FUNCTION_BLOCK FB_ParameterList // store params for permanence. THEY MUST BE PART OF AN OBJECT ELSEWHERE!
VAR
	_unNumberOfEntries : UDINT;
	_unIndexForProperties : UDINT;
	asDictionary : ARRAY[0..MAX_DICTIONARY_SIZE] OF ST_KeyReferencePair;
END_VAR
VAR CONSTANT
	MAX_DICTIONARY_SIZE : UDINT := 1000; // arbitrary
END_VAR

METHOD PUBLIC AddToList : BOOL
VAR_INPUT
	sKey : T_MaxString;
	tRef : T_Arg;
END_VAR
IF KeyExists(sKey) THEN
	RETURN;
END_IF

IF _unNumberOfEntries + 1 > MAX_DICTIONARY_SIZE THEN
	RETURN;
END_IF

asDictionary[_unNumberOfEntries].Key := sKey;
asDictionary[_unNumberOfEntries].Ref := tRef;

_unNumberOfEntries := _unNumberOfEntries + 1;

AddToList := TRUE;
END_METHOD

METHOD PUBLIC ClearList
VAR 
	indexer : UDINT;
	sBlankKeyRef : ST_KeyReferencePair;
END_VAR
FOR indexer := 0 TO _unNumberOfEntries - 1 DO
	asDictionary[indexer] := sBlankKeyRef;
END_FOR

_unNumberOfEntries := 0;
END_METHOD

METHOD PUBLIC GetByKey : T_Arg
VAR_INPUT
	sKey : STRING;
END_VAR

VAR
	indexer : UDINT;
END_VAR
FOR indexer := 0 TO _unNumberOfEntries - 1 DO
	
	IF asDictionary[indexer].Key = sKey THEN
		GetByKey := asDictionary[indexer].Ref;
		RETURN;
	END_IF;
	
END_FOR
END_METHOD

PROPERTY PUBLIC Index : UDINT
GET
Index := _unIndexForProperties;
END_GET
SET
IF Index  < _unNumberOfEntries THEN
	_unIndexForProperties := Index;
ELSE
	_unIndexForProperties := _unNumberOfEntries;
END_IF
END_SET
END_PROPERTY

PROPERTY PRIVATE IndexKey : STRING
GET // PUBLIC
IF _unIndexForProperties < _unNumberOfEntries THEN
	IndexKey := asDictionary[_unIndexForProperties].Key;
END_IF;
END_GET
END_PROPERTY

PROPERTY PRIVATE IndexRef : T_Arg
GET // PUBLIC
IF _unIndexForProperties < _unNumberOfEntries THEN
	IndexRef := asDictionary[_unIndexForProperties].Ref;
END_IF;
END_GET
END_PROPERTY

METHOD PUBLIC KeyExists : BOOL
VAR_INPUT
	sKey : T_MaxString;
END_VAR
KeyExists := NOT(F_ARGISZERO(GetByKey(sKey)));
END_METHOD

{warning 'add FB_.ParameterList.RemoveByIndex implementation'}
METHOD RemoveByIndex : BOOL
VAR_INPUT
	unListEntry : UDINT;
END_VAR
END_METHOD

{warning 'add FB_.ParameterList.RemoveByKey implementation'}
METHOD RemoveByKey : BOOL
VAR_INPUT
	sKey : T_MaxString;
END_VAR
END_METHOD

PROPERTY PUBLIC unNumberOfEntries : UDINT
GET
unNumberOfEntries := _unNumberOfEntries;
END_GET
END_PROPERTY

END_FUNCTION_BLOCK

(* stored: Version 1.1.0.1, ProductVersion 3.1.4020.12
   POU FB_ParameterList: Id {3f9645d7-6387-4cd5-895d-f3c9df1ec9bd}, SpecialFunc None
   Method AddToList: Id {d05a8a52-c1d6-4e36-b214-7645d6c4eaf0}
   Method ClearList: Id {6f827b07-8f82-44ed-947b-3d6bd655006c}
   Method GetByKey: Id {06685ac5-b98f-4071-a66a-01c516768f42}
   Property Index: Id {009f4fce-e464-4d5a-9cd0-87e23737cca6}
   Get Get: Id {9f5a3d34-8b66-40c1-abef-b68b9540fbba}
   Set Set: Id {74eb379e-0e95-41f5-90e8-3125ee755ee4}
   Property IndexKey: Id {09de8396-8d5d-4a8a-b634-d98a7f39a972}
   Get Get: Id {05470053-518e-4ad1-b6a3-68749e5ce6f8}
   Property IndexRef: Id {d14235a0-ac6a-4177-8059-3e8716ceb6fc}
   Get Get: Id {fa7f3b9d-4a46-49bd-8b16-374553f20bad}
   Method KeyExists: Id {752b1774-5a23-4c01-b8a8-82d741be2047}
   Method RemoveByIndex: Id {01f75a79-2299-4f43-a88d-488087a050a4}
   Method RemoveByKey: Id {77a5373a-3da1-4c52-9767-2fd1ed6bd18e}
   Property unNumberOfEntries: Id {dbedab0d-4484-4603-b95c-bd0bd0999e01}
   Get Get: Id {e0f330d6-3631-4fb3-942e-4eb7107aa48d} *)
